TYPE EL4xx4_Data :
STRUCT
	{attribute addProperty Name "AO Outputs Channel 1"}
	AO_OutputsChannel_1 AT %Q* : INT;
	{attribute addProperty Name "AO Outputs Channel 2"}
	AO_OutputsChannel_2 AT %Q* : INT;
	{attribute addProperty Name "AO Outputs Channel 3"}
	AO_OutputsChannel_3 AT %Q* : INT;
	{attribute addProperty Name "AO Outputs Channel 4"}
	AO_OutputsChannel_4 AT %Q* : INT;
END_STRUCT
END_TYPE

(* stored: Version 1.1.0.1, ProductVersion 3.1.4024.9
   DUT EL4xx4_Data: Id {cbcdfd6e-a583-0736-01fb-b991ebbc1636} *)
